FUNCTION_BLOCK Detector_N_Drawer_Exist (* Basic FB with empty ECC *)
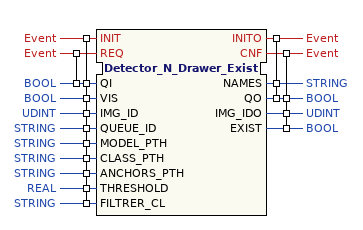
  EVENT_INPUT
    INIT WITH VIS, IMG_ID, QUEUE_ID, MODEL_PTH, CLASS_PTH, THRESHOLD, QI, ANCHORS_PTH, FILTRER_CL;
    REQ WITH QI;
  END_EVENT
  EVENT_OUTPUT
    INITO WITH QO, NAMES;
    CNF WITH QO, IMG_IDO, EXIST;
  END_EVENT
  VAR_INPUT
    QI : BOOL;
    VIS : BOOL;
    IMG_ID : UDINT;
    QUEUE_ID : STRING;
    MODEL_PTH : STRING;
    CLASS_PTH : STRING;
    ANCHORS_PTH : STRING;
    THRESHOLD : REAL;
    FILTRER_CL : STRING;
  END_VAR
  VAR_OUTPUT
    NAMES : STRING;
    QO : BOOL;
    IMG_IDO : UDINT;
    EXIST : BOOL;
  END_VAR
END_FUNCTION_BLOCK
